PROGRAM MAIN
VAR
END_VAR

PB_TestRunner();

END_PROGRAM

(* stored: Version 1.1.0.1, ProductVersion 3.1.4024.3
   POU MAIN: Id {67b9cdf5-2c90-4d9e-8b1e-7c5ddb9a41d0}, SpecialFunc None *)
